(* IEC 61131-3 sources: CODESYS-IO-Visualization/CODESYS-IO-Visualization.fbsproj/Subs, 1 file *)

(* ---- Main_ClockSync.prg.st ---- *)
PROGRAM Main_ClockSync
VAR
	SetClockTrigger: R_TRIG;
	Init: BOOL := TRUE;
END_VAR

// Set Clock Logic
SetClockTrigger(CLK := Lib_GVL.SetClock);
SetPLCClock(TZ := 'MT', DisableDST := FALSE, SetClock := SetClockTrigger.Q, SetClockValue := Lib_GVL.SetClockValue);

IF (Lib_GVL.SetClock) THEN
	Lib_GVL.SetClock := FALSE;
END_IF

//Set Globals from Library
Controller.ClockLocal := Lib_GVL.ClockLocal;
Controller.ClockUTC := Lib_GVL.ClockUTC;
